(* PLC project Tc2_Utilities.FB_FormatString Demo, tc3-libraries-kb TwinCAT 3.1 *)
(* stored: creationDateTime 2026-05-10T20:00:00, modificationDateTime 2026-05-10T20:00:00 *)

PROGRAM P_Demo_FB_FormatString
  VAR
    fbFB_FormatString : FB_FormatString;  (* Tc2_Utilities.FB_FormatString 实例 *)
    arg_sFormat : T_MaxString;  (* VAR_INPUT sFormat *)
    arg_arg1 : T_Arg;  (* VAR_INPUT arg1 *)
    arg_arg2 : T_Arg;  (* VAR_INPUT arg2 *)
    arg_arg3 : T_Arg;  (* VAR_INPUT arg3 *)
    arg_arg4 : T_Arg;  (* VAR_INPUT arg4 *)
    arg_arg5 : T_Arg;  (* VAR_INPUT arg5 *)
    arg_arg6 : T_Arg;  (* VAR_INPUT arg6 *)
    arg_arg7 : T_Arg;  (* VAR_INPUT arg7 *)
    arg_arg8 : T_Arg;  (* VAR_INPUT arg8 *)
    arg_arg9 : T_Arg;  (* VAR_INPUT arg9 *)
    arg_arg10 : T_Arg;  (* VAR_INPUT arg10 *)
    out_bError : BOOL;  (* VAR_OUTPUT bError *)
    out_nErrId : UDINT;  (* VAR_OUTPUT nErrId *)
    out_sOut : T_MaxString;  (* VAR_OUTPUT sOut *)
  END_VAR

            // ============================================================
// Tc2_Utilities.FB_FormatString 演示程序（FB 实例）
// ============================================================
// 验证步骤：
//   1. 引用 Tc2_Utilities（及依赖类型所在库 Tc2_System 等）
//   2. 编译 + 登录
//   3. 按 doc.md 给 arg_* 赋值
//   4. 在线监视 out_* / io_* 输出
// ============================================================

fbFB_FormatString(
    sFormat := arg_sFormat,
    arg1 := arg_arg1,
    arg2 := arg_arg2,
    arg3 := arg_arg3,
    arg4 := arg_arg4,
    arg5 := arg_arg5,
    arg6 := arg_arg6,
    arg7 := arg_arg7,
    arg8 := arg_arg8,
    arg9 := arg_arg9,
    arg10 := arg_arg10,
    bError => out_bError,
    nErrId => out_nErrId,
    sOut => out_sOut
);

          
END_PROGRAM
